{attribute 'linkalways'}
{attribute 'no_explicit_call' := 'do not call this POU directly'}
{attribute 'enable_dynamic_creation'}
FUNCTION_BLOCK ABSTRACT SynchronousCommand EXTENDS Disposable IMPLEMENTS I_Command;
VAR
	commandFeedback : CommandFeedback;
END_VAR

METHOD PUBLIC Abort
VAR_INPUT
END_VAR
// not possible to abort an synchonous command as the code is immediatly called in Execute()
END_METHOD

METHOD PUBLIC Execute
commandFeedback.SetBusy();

OnExecute(commandFeedback);

IF commandFeedback.Busy THEN
	commandFeedback.SetDone();
END_IF
END_METHOD

PROPERTY PUBLIC Feedback : I_CommandFeedback
GET
Feedback := commandFeedback;
END_GET
END_PROPERTY

METHOD PROTECTED ABSTRACT OnExecute
VAR_INPUT
	CommandState : I_SynchronousCommandBusyState;
END_VAR
END_METHOD

END_FUNCTION_BLOCK

(* stored: Version 1.1.0.1, ProductVersion 3.1.4024.11
   POU SynchronousCommand: Id {7933fc53-0bdf-4661-ad67-064c255651ac}, SpecialFunc None
   Folder Abstract: Id {ebbeac00-4ca1-47a4-8734-e2237b5a0ef7}
   Method Abort: Id {b2e517b9-7919-465e-971d-7a67b23f060e}
   Method Execute: Id {612fe777-3f85-448c-8eb4-857e8d26ae95}
   Property Feedback: Id {b3b0f557-629d-420a-9ab4-eed727e389a2}
   Get Get: Id {5ad12640-51ff-409c-bb11-1abdac2f96bd}
   Method OnExecute: Id {c9ca19ff-2ba5-4f6f-acc3-d35fa83ce1a8} *)
